RoboDK station: RoboDKSIM.rdk

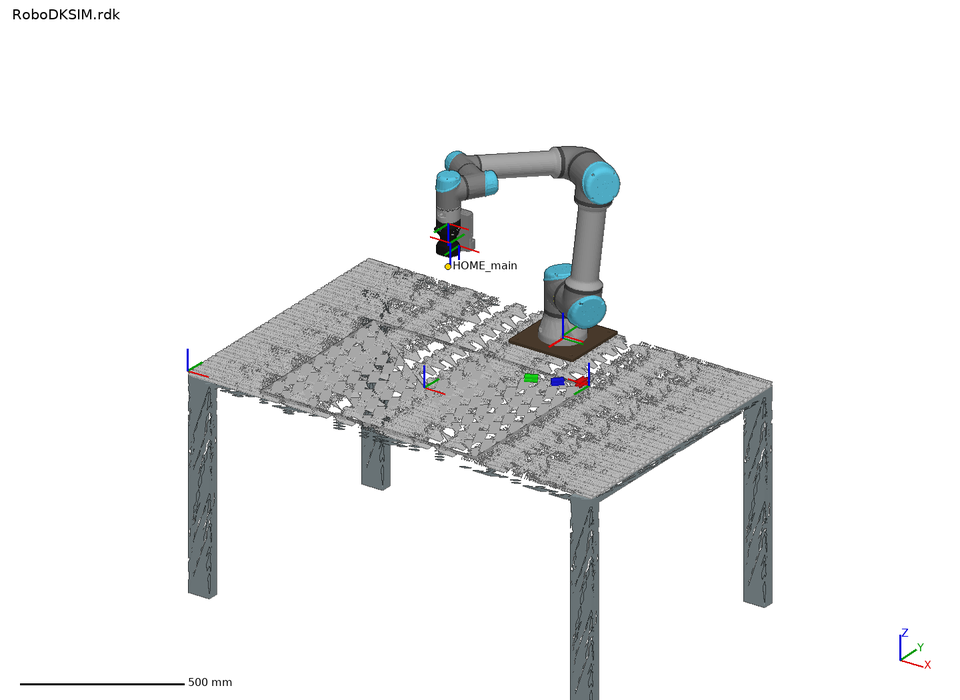
[picture v0: the station drawn from its stored meshes, robots at their saved joint values, targets as dots, program paths as lines]
Station RoboDKSIM (saved by RoboDK 5.9.4). Poses are relative to the parent item; angles as X-Y-Z fixed-axis rotations.
Station parameters (name, value as stored): PATH_MATLAB, C:\BRO_IRO_LAB\bro_iro_3_visionpnp-WS2023\files, IO_5, 1, IO_7, 1, RUN_MODE, 0, PATH_MATLAB_IMAGES, C:\BRO_IRO_LAB\bro_iro_3_visionpnp-WS2023\files\Images\, Palletizing Plugin
  - frame table_frame at (0, 1000, 0) mm
    - object table_object at (0, 0, 0) mm, size 1500 x 960.1 x 750 mm, geometry from Table.sld
    - frame white_frame at (670, 300, 10) mm
      - object white_object at (0, 0, 0) mm, size 800 x 600 x 10 mm, geometry from White Plate.STEP
    - frame robot_plate_frame at (806, 840, 0) mm, rotated rx 0 ry 0 rz -90 deg
      - object robot_plate_object at (0, 0, 0) mm, size 240 x 240 x 10 mm, 12 curves, geometry from 200731_v2_ur5e_bodenplatte_cad_jt.igs
    - frame UR5e Base at (806, 840, 10) mm
      - robot UR5e: 6 axes, payload 5 kg, reach 850 mm, repeatability 0.03 mm, weight 18.4 kg
          modified DH rows (alpha deg, a mm, theta deg, d mm): 0, 0, 0, 162.5; 90, 0, 180, 0; 0, 425, 0, 0; 0, 392.25, 0, 133.3; -90, 0, 0, 99.7; 90, 0, 180, 99.6
          joint limits [-360, -360, -360, -360, -360, -360] to [360, 360, 360, 360, 360, 360]; home [0, -90, -90, 0, 90, 0]; saved at [58.945, -96.373, 88.637, 277.652, -89.996, 328.983]
        - frame gripper_frame at (0, 0, 12) mm, rotated rx 0 ry 0 rz 180 deg
          - object Hand-E_IO_Coupling at (0, 0, -8) mm, size 75 x 105.3 x 17 mm, geometry from Hand-E_IO_Coupling.STEP
          - frame RobotiQ Hand-E Gripper Base at (0, 0, 0) mm
            - robot RobotiQ Hand-E Gripper: 1 axes
                joint limits [0] to [50]; home [0]; saved at [50]
        - frame old___camera_frame_k4a at (0, 58, 111) mm, rotated rx 0 ry 0 rz 180 deg
          - object 2203___kamerahalterung at (0, 0, 0) mm, size 103 x 46.2 x 132 mm, geometry from 2203___kamerahalterung.step
          - frame camera_frame_k4a_rgb at (-32, 0, 0) mm, rotated rx 0 ry 0 rz 180 deg
            - camera 4ka_camera_rgb_768x432
        - tool gripper_tcp, TCP at (0, 0, 158.3) mm
      - target HOME_main (Cartesian target) at (-113.59, -447.06, 379.92) mm, rotated rx -179.93 ry -0.04 rz 179.96 deg; joints [58.945, -96.373, 88.637, 277.652, -89.996, 328.983] of UR5e
    - frame gripper_move_frame at (0, 0, 0) mm
      - target open_gripper_full_target (joint target) at (692.39, 392.95, 386.22) mm, rotated rx -179.93 ry -0.04 rz 179.96 deg; joints [50, 11.333, 12.677, 10, 14.01, 14.333] of RobotiQ Hand-E Gripper
      - target open_gripper_20mm_target (Cartesian target) at (692.39, 392.95, 386.22) mm, rotated rx -179.93 ry -0.04 rz 179.96 deg; joints [20, 0, 0, 0, 0, 0] of RobotiQ Hand-E Gripper
      - target close_gripper_full_target (joint target) at (692.39, 392.95, 386.22) mm, rotated rx -179.93 ry -0.04 rz 179.96 deg; joints [0, 0, 0, 0, 0, 0] of RobotiQ Hand-E Gripper
    - frame WORLD_FRAME at (1070.19, 599.86, 10.71) mm, rotated rx 0 ry 0 rz -180 deg
      - object red_object at (19.92, 9.89, 20) mm, rotated rx 180 ry 0 rz 89.72 deg, size 40 x 20 x 20 mm, 1 curves, geometry from part.sld
      - object green_object at (161.47, 75.21, 20) mm, rotated rx 180 ry 0 rz 26.98 deg, size 40 x 20 x 20 mm, 1 curves, geometry from part.sld
      - object blue_object at (81.3, 49.51, 20) mm, rotated rx 180 ry 0 rz 47.37 deg, size 40 x 20 x 20 mm, 1 curves, geometry from part.sld
  - folder program
    - folder robodk_code
      - folder gripper_programs
        - program HandE_CLOSE_SIM (1 instructions, listed below)
        - program HandE_OPEN_SIM (1 instructions, listed below)
        - program HandE_OPEN_SIM_20mm (1 instructions, listed below)
        - program HandE_OPEN_DIO (3 instructions, listed below)
        - program HandE_CLOSE_DIO (3 instructions, listed below)
        - program Hand-E_DO_ACTIVATE (9 instructions, listed below)
      - program UR5e_HOME_SIM (3 instructions, listed below)
      - program UR5e_HOME_REL (3 instructions, listed below)

--- program HandE_CLOSE_SIM (robot RobotiQ Hand-E Gripper) ---
  MoveJ (close_gripper_full_target)

--- program HandE_OPEN_SIM (robot RobotiQ Hand-E Gripper) ---
  MoveJ (open_gripper_full_target)

--- program HandE_OPEN_SIM_20mm (robot RobotiQ Hand-E Gripper) ---
  MoveJ (open_gripper_20mm_target)

--- program HandE_OPEN_DIO (robot UR5e) ---
  Call HandE_OPEN_SIM
  Set IO_6=1
  Pause 1.0 s

--- program HandE_CLOSE_DIO (robot UR5e) ---
  Call HandE_OPEN_SIM_20mm
  Set IO_6=0
  Pause 1.0 s

--- program Hand-E_DO_ACTIVATE (robot UR5e) ---
  Call HandE_CLOSE_SIM
  Set IO_6=1
  Pause 20 ms
  Set IO_6=0
  Pause 20 ms
  Set IO_7=1
  Pause 20 ms
  Set IO_7=0
  Pause 2.0 s

--- program UR5e_HOME_SIM (robot UR5e) ---
  Set Ref.: ur5e_frame -> UR5e Base
  Set Tool: gripper_tcp
  MoveJ (Target 1) -> target HOME_main

--- program UR5e_HOME_REL (robot UR5e) ---
  Set Ref.: ur5e_frame -> UR5e Base
  Set Tool: gripper_tcp
  MoveJ (Target 1) -> target HOME_main
